FUNCTION_BLOCK FB_MotionBacklashCompensation
VAR_IN_OUT
    stMotionStage: ST_MotionStage;
END_VAR
VAR_INPUT
    bHoming: BOOL;
    bMove: BOOL;
END_VAR
VAR_OUTPUT
    bEnabled: BOOL;
    bBusy: BOOL;
    bError: BOOL;
    nErrorID: UDINT;
END_VAR
VAR
    fbBacklashCompensation: MC_BacklashCompensation;
    // Default: Positive backlash compensation
    bPrevCompensation : LREAL := 0.0;
    bBacklashCompEnable: BOOL;
END_VAR

(*Note: Configure within the axis parameters set "position correction" to true *)
(*Directional change for compensation
  default: positive backlash):
  TRUE -> Negative backlash compensation *)
(* Reset Compensation to register a new value change*)
bBacklashCompEnable R= bHoming OR (stMotionStage.fBacklashCompensation<>bPrevCompensation);
bBacklashCompEnable S= bMove;

fbBacklashCompensation(Axis:=stMotionStage.Axis,
    Enable:= ( stMotionStage.bUserBacklashEn AND bBacklashCompEnable),
    Backlash:=stMotionStage.fBacklashCompensation,
    CompensationInPositiveDirection:=(stMotionStage.fBacklashCompensation<0.0),
    Ramp:=stMotionStage.fVelocity,
    DisableMode:=DisableModeHold,
    Enabled=> stMotionStage.bBacklashStatus,
    Error=>bError,
    ErrorID=>nErrorID,
    CurrentBacklash=>stMotionStage.fCurrentBacklashCompensation);

bPrevCompensation:=stMotionStage.fBacklashCompensation;

END_FUNCTION_BLOCK

(* stored: Version 1.1.0.1
   POU FB_MotionBacklashCompensation: Id {8a5f8930-cc79-4651-8951-8645e0708394}, SpecialFunc None *)
